(* IEC 61131-3 sources: axopen.templates/axopen.template.simple/ax/src/Units/Cu10/Data/_managers_, 4 files *)

(* ---- ProcessDataExchange.st ---- *)
NAMESPACE axosimple.Cu10
    USING axosimple;
    USING AXOpen.Data;
    USING AXOpen.Core;
    USING System.Strings;

    {S7.extern=ReadWrite}
    CLASS ProcessDataExchange
        EXTENDS AXOpen.Data.AxoDataExchange
        VAR PUBLIC
            {#ix-generic:TOnline}
            {#ix-generic:TPlain as POCO}
            {#ix-attr:[AXOpen.Data.AxoDataEntityAttribute]}
            {#ix-attr:[Container(Layout.Stack)]}
            {#ix-set:AttributeName = "<#Cu10#>"}
            Payload : ProcessDataPayload;
        END_VAR
    END_CLASS
END_NAMESPACE

(* ---- ProcessDataManger.st ---- *)
NAMESPACE axosimple.Cu10
    USING axosimple;
    USING AXOpen.Data;
    USING AXOpen.Core;
    USING System.Strings;

    {S7.extern=ReadWrite}
    CLASS ProcessDataManager
        EXTENDS AXOpen.Data.AxoDataFragmentExchange
        VAR PUBLIC
            {#ix-attr:[AXOpen.Data.AxoDataFragmentAttribute]}
            Shared : axosimple.SharedDataExchange;
            {#ix-attr:[AXOpen.Data.AxoDataFragmentAttribute]}
            Data : ProcessDataExchange;
        END_VAR
    END_CLASS
END_NAMESPACE

(* ---- TechnologyDataExchange.st ---- *)
NAMESPACE axosimple.Cu10
    USING axosimple;
    USING AXOpen.Data;
    USING AXOpen.Core;
    USING System.Strings;

    {S7.extern=ReadWrite}
    CLASS TechnologyDataExchange
        EXTENDS AXOpen.Data.AxoDataExchange
        VAR PUBLIC
            {#ix-generic:TOnline}
            {#ix-generic:TPlain as POCO}
            {#ix-attr:[AXOpen.Data.AxoDataEntityAttribute]}
            {#ix-attr:[Container(Layout.Stack)]}
            {#ix-set:AttributeName = "<#Cu10#>"}
            Payload : TechnologyDataPayload;
        END_VAR
    END_CLASS
END_NAMESPACE

(* ---- TechnologyDataManager.st ---- *)
NAMESPACE axosimple.Cu10
    USING axosimple;
    USING AXOpen.Data;
    USING AXOpen.Core;
    USING System.Strings;

    {S7.extern=ReadWrite}
    CLASS TechnologyDataManager
        EXTENDS AXOpen.Data.AxoDataFragmentExchange
        VAR PUBLIC
            {#ix-attr:[AXOpen.Data.AxoDataFragmentAttribute]}
            Shared : axosimple.TechnologySharedDataExchange;
            {#ix-attr:[AXOpen.Data.AxoDataFragmentAttribute]}
            Data : TechnologyDataExchange;
        END_VAR
    END_CLASS
END_NAMESPACE
